TYPE TcoVisionData :
STRUCT	
	Length : UINT;
	Data : ARRAY[0..TcoVisionParams.MAX_BYTE_ARRAY] OF BYTE;
END_STRUCT
END_TYPE

(* stored: Version 1.1.0.1, ProductVersion 3.1.4024.11
   DUT TcoVisionData: Id {994e25c9-4b0f-0e4f-00ae-28bac0eec7d4} *)
